{attribute addProperty BoxType "EL2262-0000-0002"}
{attribute addProperty Id "CycCount0AT %Q*CycCount0_307034DC1620Sample0AT %Q*ARRAY[0..9] OF Sample_ABF5BEA980100GapAT %Q*EMPTY_STRUCTURE000CycCount1AT %Q*CycCount1_7787FA1D1620Sample1AT %Q*ARRAY[0..9] OF Sample_4351E8AC80100Gap_1AT %Q*EMPTY_STRUCTURE000WcStateAT %I*WcState_28A8677510.1250InfoDataAT %I*InfoData_7231B2DD80100"}
{attribute addProperty CRC "3244892927"}
{attribute addProperty SizeInBites "273"}
{attribute addProperty SizeInBytes "34.125"}
TYPE EL2262_131C31B2 :
STRUCT
	{attribute addProperty Name "CycCount0"}
	CycCount0 : CycCount0_307034DC;
	{attribute addProperty Name "Sample0"}
	Sample0 : ARRAY[0..9] OF Sample_ABF5BEA9;
	{attribute addProperty Name "Gap"}
	Gap : EMPTY_STRUCTURE;
	{attribute addProperty Name "CycCount1"}
	CycCount1 : CycCount1_7787FA1D;
	{attribute addProperty Name "Sample1"}
	Sample1 : ARRAY[0..9] OF Sample_4351E8AC;
	{attribute addProperty Name "Gap_1"}
	Gap_1 : EMPTY_STRUCTURE;
	{attribute addProperty Name "WcState"}
	WcState : WcState_28A86775;
	{attribute addProperty Name "InfoData"}
	InfoData : InfoData_7231B2DD;
END_STRUCT
END_TYPE

(* stored: Version 1.2.0.0, ProductVersion 3.1.4024.9
   DUT EL2262_131C31B2: Id {46deb77e-fb51-43f7-93d5-d2f172dd3334} *)
